Fanuc KAREL source: kt00033.KL

-- PROVISIONAL review KL for V770-1; original PC SHA256 f1fdfeda29697f31eb35a1f037fdb114c82d0319819b2d48fb440714266557d5
-- Incomplete behavior may be omitted. Consult companion uncertainty JSON. Do not deploy.
PROGRAM KT00033
%NOLOCKGROUP
VAR
  I1 : INTEGER
  I2 : INTEGER
  OUT : INTEGER
BEGIN
  -- UNRESOLVED_PC offsets 5-16; opcodes 2E,23
  -- UNRESOLVED_PC offsets 21-32; opcodes 2E,23
  -- UNRESOLVED_PC offsets 37-48; opcodes 2E,23
  -- UNRESOLVED_PC offsets 53-64; opcodes 2E,23
  -- UNRESOLVED_PC offsets 69-88; opcodes 21,21,53,23
  -- UNRESOLVED_PC offsets 93-97; opcodes 7F
END KT00033
